FUNCTION_BLOCK FB_BMS_IO

VAR_INPUT
	HWControl			:	st_BMS_IO;
END_VAR

VAR_OUTPUT
	BMSPowerControl			AT %Q* : st_BMS_IO;
END_VAR

VAR
	PowerUpDelay	:	TON := (PT := TIME#1s0ms);
END_VAR


BMSPowerControl.b_BMS_230V_Enable := HWControl.b_BMS_230V_Enable;
BMSPowerControl.b_BMS_24V_Enable	:= HWControl.b_BMS_24V_Enable;

END_FUNCTION_BLOCK

(* stored: Version 1.1.0.1, ProductVersion 3.1.4024.12
   POU FB_BMS_IO: Id {09c82cc6-0e1a-4de8-8d19-79768c652534}, SpecialFunc None *)
